FUNCTION_BLOCK CL_AxisDriverL1LeftFront EXTENDS CL_AxisDriverAX8206
VAR
END_VAR

SUPER^();

METHOD PUBLIC Init : BOOL
VAR_INPUT  
  stDriver : POINTER TO ST_DriverAX8206_HWI;
END_VAR
Init := FALSE;
IF stDriver <> 0 THEN
  Init := SUPER^.InitDriver(stDriverCom_P := ADR(stDriver^.comState), stDriverCh_P := ADR(stDriver^.stFront));
END_IF
END_METHOD

METHOD PROTECTED InitDefect : BOOL
VAR_INPUT
END_VAR
InitDefect := SUPER^.InitDefect();
ADSLOGSTR(ADSLOG_MSGTYPE_LOG, 'CL_AxisDriverL1LeftFront init defect','');
END_METHOD

END_FUNCTION_BLOCK

(* stored: Version 1.1.0.1, ProductVersion 3.1.4024.12
   POU CL_AxisDriverL1LeftFront: Id {200b1fcd-14b8-4d99-97a7-7230d8a0e054}, SpecialFunc None
   Method Init: Id {33cfbbe0-1d43-4519-95be-cc28fab85ad1}
   Method InitDefect: Id {53bcca80-abde-4b94-96ae-a94cd40d2c69} *)
